DATA_BLOCK "ST10_SystemModeFB_iDB"
{ S7_Optimized_Access := 'TRUE' }
VERSION : 0.1
NON_RETAIN
// ATTRIBUTES
// AUTO_NUMBER = False
// BLOCK_NUMBER = 1000
// END_ATTRIBUTES
"SystemMode"

BEGIN

END_DATA_BLOCK

